FUNCTION_BLOCK SkillMessage (* Basic FB with empty ECC *)
  (* Standard: 61499-2 *)
  (* Version 1.0, 2021-03-18, dummy *)
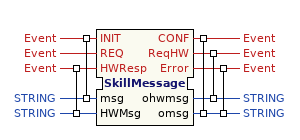
  EVENT_INPUT
    INIT WITH msg;
    REQ;
    HWResp WITH HWMsg;
  END_EVENT
  EVENT_OUTPUT
    CONF WITH omsg;
    ReqHW WITH ohwmsg;
    Error WITH omsg;
  END_EVENT
  VAR_INPUT
    msg : STRING;
    HWMsg : STRING;
  END_VAR
  VAR_OUTPUT
    ohwmsg : STRING;
    omsg : STRING;
  END_VAR
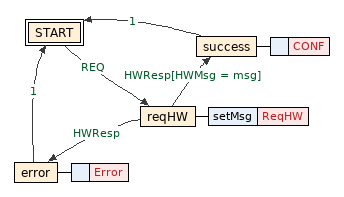
  EC_STATES
    START; (* Initial State *)
    reqHW : setMsg -> ReqHW;
    success : -> CONF;
    error : -> Error;
  END_STATES
  EC_TRANSITIONS
    START TO reqHW := REQ;
    reqHW TO success := HWResp[HWMsg = msg];
    reqHW TO error := HWResp;
    error TO START := 1;
    success TO START := 1;
  END_TRANSITIONS
  ALGORITHM setMsg IN ST:
omsg := msg;
  END_ALGORITHM
  ALGORITHM setErrorMsg IN ST:
omsg := HWMsg;
  END_ALGORITHM
END_FUNCTION_BLOCK
